FUNCTION_BLOCK FB_DRIVE_MSG_LOG
VAR
	Buffer	: ARRAY[0..MaxBufferSize] OF ST_DRIVE_MSG;
	Index : INT;
END_VAR
VAR CONSTANT
	MaxBufferSize	: INT := 1000;
END_VAR

METHOD AddMsg : BOOL
VAR_INPUT
	TimeStamp			: DT;
	LeftVelocity		: INT;
	RightVelocity		: INT;
	LeftSteeringAngle	: LREAL;
	RightSteeringAngle	: LREAL;
	LeftCurrent			: REAL;
	RightCurrent		: REAL;
	LeftStatusCode		: UINT;
	RightStatusCode		: UINT;
END_VAR
VAR
	i: INT;
END_VAR
FOR i := 0 TO MaxBufferSize DO
	IF Buffer[MaxBufferSize - i].LeftVelocity = 0.0 THEN
		CONTINUE;
	ELSE
		Buffer[MaxBufferSize - i + 1].TimeStamp 			:= Buffer[MaxBufferSize - i].TimeStamp;
		Buffer[MaxBufferSize - i + 1].LeftVelocity 			:= Buffer[MaxBufferSize - i].LeftVelocity;
		Buffer[MaxBufferSize - i + 1].RightVelocity 		:= Buffer[MaxBufferSize - i].RightVelocity;
		Buffer[MaxBufferSize - i + 1].LeftSteeringAngle 	:= Buffer[MaxBufferSize - i].LeftSteeringAngle;
		Buffer[MaxBufferSize - i + 1].RightSteeringAngle 	:= Buffer[MaxBufferSize - i].RightSteeringAngle;
		Buffer[MaxBufferSize - i + 1].LeftCurrent 			:= Buffer[MaxBufferSize - i].LeftCurrent;
		Buffer[MaxBufferSize - i + 1].RightCurrent 			:= Buffer[MaxBufferSize - i].RightCurrent;
		Buffer[MaxBufferSize - i + 1].LeftStatusCode 		:= Buffer[MaxBufferSize - i].LeftStatusCode;
		Buffer[MaxBufferSize - i + 1].RightStatusCode 		:= Buffer[MaxBufferSize - i].RightStatusCode;
	END_IF
END_FOR

Buffer[0].Timestamp 			:= TimeStamp;
Buffer[0].LeftVelocity 			:= LeftVelocity;
Buffer[0].RightVelocity 		:= RightVelocity;
Buffer[0].LeftSteeringAngle 	:= LeftSteeringAngle;
Buffer[0].RightSteeringAngle 	:= RightSteeringAngle;
Buffer[0].LeftCurrent 			:= LeftCurrent;
Buffer[0].RightCurrent 			:= RightCurrent;
Buffer[0].LeftStatusCode 		:= LeftStatusCode;
Buffer[0].RightStatusCode 		:= RightStatusCode;

Index := Index + 1;
END_METHOD

END_FUNCTION_BLOCK

(* stored: Version 1.1.0.1, ProductVersion 3.1.4024.12
   POU FB_DRIVE_MSG_LOG: Id {273aa02f-b17c-4960-9963-8a7c0add0e7b}, SpecialFunc None
   Method AddMsg: Id {4c6b5223-b671-431a-885e-811c84482326} *)
